FUNCTION_BLOCK FB_ServingCustomer IMPLEMENTS I_State
VAR_INPUT
	(* Pointer to the ATM Machine*)
	pATM_Machine	: POINTER TO FB_ATM_Machine;
END_VAR
VAR_OUTPUT
END_VAR
VAR
END_VAR

METHOD Cancel : BOOL
ADSLOGSTR(ADSLOG_MSGTYPE_LOG, 'Transaction canceled, going to idle...', '');
pATM_Machine^.SetState(pATM_Machine^.IdleState);
END_METHOD

METHOD Card_Ejected : BOOL
ADSLOGSTR(ADSLOG_MSGTYPE_LOG, 'Card has been ejected, going to idle...', '');
pATM_Machine^.SetState(pATM_Machine^.IdleState);
END_METHOD

METHOD Card_Inserted : BOOL
END_METHOD

PROPERTY Description : E_StateDescription
GET
Description := E_StateDescription.ServingCustomer;
END_GET
END_PROPERTY

METHOD Failure : BOOL
ADSLOGSTR(ADSLOG_MSGTYPE_LOG, 'Transaction failed, contact service...', '');
pATM_Machine^.SetState(pATM_Machine^.OutOfServiceState);
END_METHOD

METHOD FB_Init : BOOL
VAR_INPUT
	(* if TRUE, the retain variables are initialized (warm start / cold start)*)
	bInitRetains	: BOOL;
	(* if TRUE, the instance afterwards gets moved into the copy code (online change)*)
	bInCopyCode	: BOOL;
	(* Pointer to the ATM Machine*)
	pATM_Machine	: POINTER TO FB_ATM_Machine;
END_VAR
THIS^.pATM_Machine := pATM_Machine;
END_METHOD

METHOD Op : BOOL
END_METHOD

METHOD Service : BOOL
END_METHOD

METHOD SystemTest_OK : BOOL
END_METHOD

METHOD Turn_Off : BOOL
END_METHOD

METHOD Turn_On : BOOL
END_METHOD

END_FUNCTION_BLOCK

(* stored: Version 1.1.0.1, ProductVersion 3.1.4024.12
   POU FB_ServingCustomer: Id {2169bdb5-0da4-0ea5-24fe-5fde7652ce39}, SpecialFunc None
   Method Cancel: Id {0e0fe738-b3e9-0358-2d81-02f6cd38afb2}
   Method Card_Ejected: Id {747865e4-dec6-08e9-384e-b8fa1a87fd13}
   Method Card_Inserted: Id {496c6b96-2532-0095-24e3-1ab072d73dc9}
   Property Description: Id {8489062d-1154-04dd-1950-3fc62e92bac3}
   Get Get: Id {a852d8cb-c913-00cf-3bf9-dc37610b440f}
   Method Failure: Id {aeaf7ee5-2b0b-09ab-1796-fa68bbf06b98}
   Method FB_Init: Id {f7335f31-dc20-01dd-07c2-500833277a92}
   Method Op: Id {9249b1da-093c-0417-3d7d-fb694f350cc8}
   Method Service: Id {6fbae138-be53-0222-29db-22d42af02186}
   Method SystemTest_OK: Id {058fed9a-4cbb-0ced-299f-a0df271f8cd4}
   Method Turn_Off: Id {f7a7925a-d73d-0675-1999-5077c1979473}
   Method Turn_On: Id {fdac9bf2-2e0e-06f4-364f-b3e5cdb12bf2} *)
